(*
SPDX-FileCopyrightText: © 2026 Oleksandr Tiutyk <trofimich@gmail.com>
SPDX-License-Identifier: MIT
License: https://opensource.org/license/mit
*)

(*!
<summary>Holds at most 255 flattened entries. Inner exception graphs must be acyclic.</summary>
<description>
Self-add is forbidden by contract; no recursive graph validation is performed.
</description>
*)

{attribute 'enable_dynamic_creation'}	
{attribute 'no_explicit_call' := 'do not call this function block directly'} 


FUNCTION_BLOCK AggregateException EXTENDS Exception IMPLEMENTS IAggregateException
VAR
	{attribute 'hide'} 
	_ClassName : STRING := __POUNAME();
	
	_InnerExceptions : POINTER TO IException;
	{attribute 'hide'} 
	_InnerExceptionCount : UINT;
END_VAR
VAR CONSTANT
	MAX_INNER_EXCEPTION_COUNT : UINT := 255;
END_VAR

(*!
<summary>Flattens aggregates; borrows dynamic inners and clones static inners for automatic cleanup.</summary>
<description>
Owns only the reference array. Allocation failure uses the shared fatal memory latch.
Do not pass THIS or a cyclic exception graph. Null/empty aggregate inputs add nothing.
Exceeding 255 entries raises latched OUT_OF_MEMORY before preparing the next entry.
Flattening is incremental: prior successful additions are not rolled back on failure.
</description>
*)

METHOD AddInnerException
VAR_INPUT
	innerException : IException; 
END_VAR
VAR
	aggregateException : IAggregateException;
	i : DINT;
	subInnerException : IException;	
	
	newInnerExceptionArray : POINTER TO IException;
	preparedInnerException : IException;
END_VAR
IF innerException = 0 THEN
	RETURN;
END_IF

IF __QUERYINTERFACE(innerException, aggregateException) THEN
	FOR i := 0 TO TO_DINT(aggregateException.InnerExceptionCount) - 1 DO
		subInnerException := aggregateException.GetInnerException(i);
		
		AddInnerException(subInnerException);
	END_FOR
ELSE
	IF _InnerExceptionCount >= MAX_INNER_EXCEPTION_COUNT THEN
		DynamicMemoryManager.RaiseAllocationFailure();
		RETURN;
	END_IF

	// Prepare the inner before replacing any existing array storage.
	IF innerException.IsDynamicInstance THEN
		preparedInnerException := innerException;
	ELSE
		__QUERYINTERFACE(innerException.Clone(), preparedInnerException);
	END_IF

	newInnerExceptionArray := __NEW(POINTER TO IException, (_InnerExceptionCount + 1));
	IF newInnerExceptionArray = 0 THEN
		DynamicMemoryManager.RaiseAllocationFailure();
		RETURN;
	END_IF
		
	IF _InnerExceptionCount > 0 THEN
		Tc2_System.MEMCPY(newInnerExceptionArray, _InnerExceptions, TO_UDINT(XSIZEOF(POINTER TO IException) * _InnerExceptionCount));	
	
		__DELETE(_InnerExceptions);
	END_IF
		
	newInnerExceptionArray[_InnerExceptionCount] := preparedInnerException;
	
	_InnerExceptions := newInnerExceptionArray; 
	_InnerExceptionCount := _InnerExceptionCount + 1;
END_IF
END_METHOD

{attribute 'monitoring' := 'call'}
PROPERTY ClassName : REFERENCE TO STRING
GET
ClassName REF= _ClassName;
END_GET
END_PROPERTY

(*!
<summary>Releases the owned reference array and resets metadata; does not delete borrowed inners.</summary>
<description>
Repeated Clear is allowed.
</description>
*)

METHOD Clear
IF _InnerExceptions <> 0 THEN
	__DELETE(_InnerExceptions);
END_IF

_InnerExceptionCount := 0;

SUPER^.Clear();
END_METHOD

(*!
<summary>Returns a distinct auto-disposed aggregate with copied metadata and its own reference array.</summary>
<description>
Empty aggregates also produce a distinct empty clone; dynamic inners remain borrowed.
</description>
*)

METHOD Clone : IObject
VAR
	exceptionClone : POINTER TO AggregateException;
		
	i : DINT;
END_VAR
exceptionClone := __NEW(AggregateException);

IF exceptionClone = 0 THEN
	DynamicMemoryManager.RaiseAllocationFailure();
	RETURN;
END_IF

exceptionClone^.SourceFullPOUName := _SourceFullPOUName;
exceptionClone^.SourcePosition := _SourcePosition;
exceptionClone^.LocalTimestamp := _LocalTimestamp;	
exceptionClone^.UtcTimestamp := _UtcTimestamp;	

FOR i := 0 TO TO_DINT(_InnerExceptionCount) - 1 DO
	exceptionClone^.AddInnerException(GetInnerException(i));
END_FOR

Clone := exceptionClone^;
END_METHOD

(*!
<summary>Destination must be empty and distinct from source. This helper does not clear existing entries.</summary>
<description>
Copies metadata and adds source entries using AddInnerException's ownership rules.
</description>
*)

METHOD PROTECTED CopyFields
VAR_IN_OUT CONSTANT
	sourceExxception : AggregateException;	
END_VAR
VAR
	i : DINT;
END_VAR
_SourceFullPOUName := sourceExxception.SourceFullPOUName;
_SourcePosition := sourceExxception.SourcePosition;
_LocalTimestamp := sourceExxception.LocalTimestamp;	
_UtcTimestamp := sourceExxception.UtcTimestamp;	

FOR i := 0 TO TO_DINT(sourceExxception.InnerExceptionCount) - 1 DO
	AddInnerException(sourceExxception.GetInnerException(i));
END_FOR
END_METHOD

{attribute 'monitoring' := 'call'}
PROPERTY Empty : BOOL
GET
Empty := _InnerExceptionCount = 0;
END_GET
END_PROPERTY

//!<param name="bInCopyCode">if TRUE, the exit method is called for exiting an instance that is copied afterwards (online change).</param>

METHOD FB_exit : BOOL
VAR_INPUT
	
	bInCopyCode	: BOOL;
END_VAR
Clear();
END_METHOD

METHOD GetInnerException : IException
VAR_INPUT
	index : DINT;
END_VAR
IF index >= 0 AND_THEN index < _InnerExceptionCount THEN
	GetInnerException := _InnerExceptions[index];
END_IF
END_METHOD

(*!
<summary>With default options an empty aggregate returns "0 aggregated exceptions".</summary>
*)

METHOD GetMessage : ERROR_MESSAGE
VAR_INPUT
	showSource : BOOL := FALSE;
	timestampDisplayMode : TIMESTAMP_DISPLAY_MODE := TIMESTAMP_DISPLAY_MODE.HIDDEN;
END_VAR
VAR
	stringBuilder : WideStringBuilder;
	
	i : DINT;
	innerException : IException;
	innerExceptionMessage : ERROR_MESSAGE;
END_VAR
stringBuilder
	.Append(_InnerExceptionCount)
	.AppendString(Exceptions.AGGREGATE_EXCEPTION_SUFFIX);

IF timestampDisplayMode <> TIMESTAMP_DISPLAY_MODE.HIDDEN THEN
	stringBuilder.AppendString(Exceptions.TIME_PREFIX);
	AppendTimestampDescription(stringBuilder, timestampDisplayMode, _LocalTimestamp, _UtcTimestamp);
END_IF

IF showSource THEN
	stringBuilder
		.AppendString(Exceptions.SOURCE_PREFIX)
		.AppendString255(TO_WSTRING(_SourceFullPOUName))
		.AppendStringIf(Exceptions.SOURCE_POSITION_PREFIX, sourcePosition <> '')
		.AppendString255If(TO_WSTRING(sourcePosition), sourcePosition <> '');
END_IF

FOR i := 0 TO TO_DINT(_InnerExceptionCount) - 1 DO
	innerException := _InnerExceptions[i];
	
	innerExceptionMessage := innerException.GetMessage(showSource, timestampDisplayMode);
	
	stringBuilder
		.AppendString255(WideStrings.NewLine)
		.Append(i)
		.AppendString(Exceptions.MESSAGE_NUMBER_SUFFIX)	
		.AppendString(" ")
		.Append(innerExceptionMessage);
END_FOR		

stringBuilder.AssignToString(GetMessage);
END_METHOD

METHOD FINAL GetRootException : IException
IF _InnerExceptionCount > 0 THEN
	GetRootException := GetInnerException(0);
	
	GetRootException := GetRootException.GetRootException();
ELSE
	GetRootException := THIS^;
END_IF
END_METHOD

{attribute 'monitoring' := 'call'}
PROPERTY InnerExceptionCount : UINT
GET
InnerExceptionCount := _InnerExceptionCount;
END_GET
END_PROPERTY

{attribute 'monitoring' := 'call'}
PROPERTY NamespaceName : REFERENCE TO STRING
GET
NamespaceName REF= CurrentNamespace.Name;
END_GET
END_PROPERTY

{attribute 'monitoring' := 'call'}
PROPERTY SelfSize : ULINT
GET
SelfSize := XSIZEOF(THIS^);
END_GET
END_PROPERTY

METHOD Throw
VAR_INPUT
	sourceNamespaceName : STRING;
	sourceClassName : STRING;
	sourcePOUName : STRING;
	sourcePosition : STRING;
END_VAR
_SourceFullPOUName := GetFullPOUName(sourceNamespaceName, sourceClassName, sourcePOUName);
_SourcePosition := sourcePosition;
_LocalTimestamp := System.SystemLocalDateTime;
_UtcTimestamp := System.SystemUtcDateTime;

ExceptionManager.Throw(THIS^);
END_METHOD

METHOD ToError
VAR_IN_OUT CONSTANT
	targetError : ERROR;
END_VAR
VAR_INPUT
	severity : ERROR_SEVERITY;	
END_VAR
VAR
	rootException : IException;
END_VAR
IF NOT __ISVALIDREF(targetError) THEN
	RETURN;
END_IF

IF _InnerExceptionCount <= 0 THEN
	targetError.Fill(
		severity,
		GetSourceDescription(),
		Exceptions.UNSPECIFIED_SOURCE,
		"Empty aggregate exception (zero inner exceptions)",
		"",
		LocalTimestamp,
		UtcTimestamp
	);
	
	RETURN;
END_IF

rootException := GetInnerException(0);

targetError.Fill(
	severity,
	Strings.Concat255(TO_STRING(_InnerExceptionCount), ' exceptions occured'),
	rootException.GetSourceDescription(),
	GetMessage(),
	rootException.GetMessage(),
	LocalTimestamp,
	UtcTimestamp
);
END_METHOD

END_FUNCTION_BLOCK

(* stored: Version 1.1.0.1
   POU AggregateException: Id {8695c106-e7fb-42e2-9023-16f2aac84192}, SpecialFunc None
   Folder Service members: Id {c31ba568-bfb3-4fae-ac77-198d7130e4aa}
   Method AddInnerException: Id {bfce23ea-1373-4ba3-866d-7d8a69bbfdab}
   Property ClassName: Id {bd878664-be6a-49ac-98d9-c91ba460da65}
   Get Get: Id {998929b6-4b31-437f-a5e5-a39dd1d6dc61}
   Method Clear: Id {e4a1b8c7-9686-4ca1-8667-c1a80c4453a6}
   Method Clone: Id {486d4ff9-908c-48b8-a667-acc4326b9c0c}
   Method CopyFields: Id {0584c9e4-cd70-4feb-b915-e7d77badfcc1}
   Property Empty: Id {d2ade75f-e0d1-434c-8840-7186cc0e6f7a}
   Get Get: Id {c0b1f376-6cae-43f3-86ac-6339a2e458c0}
   Method FB_exit: Id {56b27e89-e503-4505-9d3d-a810a3015a78}
   Method GetInnerException: Id {208441ce-95c7-4cde-b727-858df1415649}
   Method GetMessage: Id {76c9ffdd-6b67-4a44-aa6c-571f736f1a93}
   Method GetRootException: Id {3947d49e-1dd5-493f-96aa-4bb6602d0186}
   Property InnerExceptionCount: Id {734e1c9b-9746-493a-8ce4-7a56d60ff952}
   Get Get: Id {d38858e5-3bfc-4ef7-a005-fb8d5b223e97}
   Property NamespaceName: Id {494a86d9-380f-42f2-920d-5159f570a5a6}
   Get Get: Id {d3864769-88da-4cdf-9783-f994cd245ebc}
   Property SelfSize: Id {174b7a67-11f4-4a03-a1cf-384fffd912fd}
   Get Get: Id {0f74268c-6818-41c3-9fc5-eec449ba75e8}
   Method Throw: Id {1b8b1f86-dba3-4290-8289-61d8dd5d28c8}
   Method ToError: Id {d4ff76fe-085d-4302-a17b-b20e40bfa8ce} *)
